INTERFACE I_Base

PROPERTY Busy : Bool
GET
END_GET
END_PROPERTY

PROPERTY Done : Bool
GET
END_GET
END_PROPERTY

PROPERTY Error : Bool
GET
END_GET
END_PROPERTY

PROPERTY ErrorID : UDINT
GET
END_GET
END_PROPERTY

END_INTERFACE

(* stored: Version 1.1.0.1, ProductVersion 3.1.4024.14
   Itf I_Base: Id {e28f02d3-80c8-4cf4-984c-d5994be10a9f}
   Folder Properties: Id {15324833-6475-461c-b2e2-23a101e1013b}
   Property Busy: Id {35a9da76-daa5-4c40-88c6-b0135733439f}
   Get Get: Id {501d2de1-9557-400a-acb6-e88767b1c569}
   Property Done: Id {52940905-09b5-41d4-a583-16de5914e142}
   Get Get: Id {bb86aeff-a68a-47ea-a1d3-5838ae8d7eb1}
   Property Error: Id {32e3bb8a-7329-4174-afef-bf324c83e960}
   Get Get: Id {d7c3d065-62c6-46d6-8259-d34b92697e61}
   Property ErrorID: Id {b10cdd15-a1b0-4247-9b95-ef52b9e30e2f}
   Get Get: Id {8de0f140-5323-494f-a596-403d956fb360} *)
